Staubli VAL3: onFunctionView.pgx

public program onFunctionView(num x_nIndex, string x_sEvent, num x_nFunctionKey)
  local string l_sMessage
  local string l_sButton[2]
  local bool l_bYes
  local tool l_tTool
  local point l_pAlign
  local string l_sMessage2
  local joint l_jJoint
  local num l_nIndexFrame
  local frame l_fFrame
begin
  //
  // do on Key action
  //
  // x_nIndex = actual index item
  // x_sEvent = actual event item
  //
  switch x_nFunctionKey
    // F1 button
    case 271
      // HERE JOINT
      if !cycleStatus:bCycle
        call language:message(l_sMessage,160)
        call language:getYesNo(l_sButton)
        // ask the yes_no question
        call use:yes_no(l_sMessage,l_sButton,l_bYes)
        if l_bYes
          call HerePoint(x_nIndex)
        endIf
      endIf
    break
    // F2 button
    case 272
      // ALIGN
      if !cycleStatus:bCycle and !cycleStatus:bSimulation
        resetMotion()
        call getFrameId(l_nIndexFrame)
        l_fFrame=saveData:fFrameItem[l_nIndexFrame].fFrame
        // tool
        call tcp:getTool(l_tTool,jEditPoint.nIndexTool)
        l_pAlign=here(l_tTool,l_fFrame)
        l_pAlign.trsf=align(l_pAlign.trsf,l_fFrame.trsf)
        // check the align
        if pointToJoint(l_tTool,herej(),l_pAlign,l_jJoint)
          call language:message(l_sMessage,203)
          call language:message(l_sMessage2,134)
          l_sMessage=l_sMessage+" "+l_sMessage2+"..."
          call use:timerDialog(l_sMessage,0)
          movel(l_pAlign,l_tTool,mMdesc)
          watch(isEmpty() or isKeyPressed(255),3)
          if !isEmpty()
            resetMotion()
          endIf
          delay(2)
        endIf
      endIf
    break
    // F3 button
    case 273
    break
    // F4 button
    case 274
    break
    // F5 button
    case 275
    break
    // F6 button
    case 276
    break
    // F7 button
    case 277
    break
    // F8 button
    case 278
    break
  endSwitch
end
